(* Logix 5000 project; controller ACMI_PLC vendor 1 type 14 code 101 rev 19.11; software revision 19.01; part 3 of 18 *)

        [755].TIME.MICROSECOND := 993025, [755].EVENT := '2016/09/22   13:48:08   USER : PPS RESET FAULT BUTTON PRESSED', [756].TIME.YEAR := 2016, [756].TIME.MONTH := 9, [756].TIME.DAY := 22, [756].TIME.HOUR := 13, [756].TIME.MINUTE := 48, [756].TIME.SECOND := 37, [756].TIME.MICROSECOND := 592455, [756].EVENT := '2016/09/22   13:48:37   FAULT : QOW1 : Charge Outside Window Detected', [757].TIME.YEAR := 2016, [757].TIME.MONTH := 9, [757].TIME.DAY := 22, [757].TIME.HOUR := 13, [757].TIME.MINUTE := 58, [757].TIME.SECOND := 51, [757].TIME.MICROSECOND := 992497, [757].EVENT := '2016/09/22   13:58:51   USER : PPS RESET FAULT BUTTON PRESSED', [758].TIME.YEAR := 2016, [758].TIME.MONTH := 9, [758].TIME.DAY := 22, [758].TIME.HOUR := 13, [758].TIME.MINUTE := 59, [758].TIME.SECOND := 13, [758].TIME.MICROSECOND := 392501, [758].EVENT := '2016/09/22   13:59:13   USER : PPS RESET FAULT BUTTON PRESSED', [759].TIME.YEAR := 2016, [759].TIME.MONTH := 9, [759].TIME.DAY := 22, [759].TIME.HOUR := 14, [759].TIME.MINUTE := 6, [759].TIME.SECOND := 54, [759].TIME.MICROSECOND := 592461, [759].EVENT := '2016/09/22   14:06:54   FAULT : QOW1 : Charge Outside Window Detected', [760].TIME.YEAR := 2016, [760].TIME.MONTH := 9, [760].TIME.DAY := 22, [760].TIME.HOUR := 14, [760].TIME.MINUTE := 6, [760].TIME.SECOND := 54, [760].TIME.MICROSECOND := 692501, [760].EVENT := '2016/09/22   14:06:54   USER : PPS RESET FAULT BUTTON PRESSED', [761].TIME.YEAR := 2016, [761].TIME.MONTH := 9, [761].TIME.DAY := 22, [761].TIME.HOUR := 14, [761].TIME.MINUTE := 9, [761].TIME.SECOND := 18, [761].TIME.MICROSECOND := 892502, [761].EVENT := '2016/09/22   14:09:18   USER : PPS RESET FAULT BUTTON PRESSED', [762].TIME.YEAR := 2016, [762].TIME.MONTH := 9, [762].TIME.DAY := 22, [762].TIME.HOUR := 14, [762].TIME.MINUTE := 9, [762].TIME.SECOND := 19, [762].TIME.MICROSECOND := 92924, [762].EVENT := '2016/09/22   14:09:19   USER : PPS RESET FAULT BUTTON PRESSED', [763].TIME.YEAR := 2016, [763].TIME.MONTH := 9,
        [763].TIME.DAY := 22, [763].TIME.HOUR := 14, [763].TIME.MINUTE := 9, [763].TIME.SECOND := 19, [763].TIME.MICROSECOND := 292500, [763].EVENT := '2016/09/22   14:09:19   USER : PPS RESET FAULT BUTTON PRESSED', [764].TIME.YEAR := 2016, [764].TIME.MONTH := 9, [764].TIME.DAY := 22, [764].TIME.HOUR := 14, [764].TIME.MINUTE := 10, [764].TIME.SECOND := 9, [764].TIME.MICROSECOND := 92519, [764].EVENT := '2016/09/22   14:10:09   USER : PPS RESET FAULT BUTTON PRESSED', [765].TIME.YEAR := 2016, [765].TIME.MONTH := 9, [765].TIME.DAY := 22, [765].TIME.HOUR := 14, [765].TIME.MINUTE := 10, [765].TIME.SECOND := 22, [765].TIME.MICROSECOND := 892490, [765].EVENT := '2016/09/22   14:10:22   FAULT : QOW1 : Charge Outside Window Detected', [766].TIME.YEAR := 2016, [766].TIME.MONTH := 9, [766].TIME.DAY := 22, [766].TIME.HOUR := 14, [766].TIME.MINUTE := 14, [766].TIME.SECOND := 58, [766].TIME.MICROSECOND := 893026, [766].EVENT := '2016/09/22   14:14:58   USER : PPS RESET FAULT BUTTON PRESSED', [767].TIME.YEAR := 2016, [767].TIME.MONTH := 9, [767].TIME.DAY := 22, [767].TIME.HOUR := 14, [767].TIME.MINUTE := 17, [767].TIME.SECOND := 16, [767].TIME.MICROSECOND := 392944, [767].EVENT := '2016/09/22   14:17:16   USER : PPS RESET FAULT BUTTON PRESSED', [768].TIME.YEAR := 2016, [768].TIME.MONTH := 9, [768].TIME.DAY := 22, [768].TIME.HOUR := 14, [768].TIME.MINUTE := 24, [768].TIME.SECOND := 16, [768].TIME.MICROSECOND := 292454, [768].EVENT := '2016/09/22   14:24:16   FAULT : QOW1 : Charge Outside Window Detected', [769].TIME.YEAR := 2016, [769].TIME.MONTH := 9, [769].TIME.DAY := 22, [769].TIME.HOUR := 14, [769].TIME.MINUTE := 24, [769].TIME.SECOND := 16, [769].TIME.MICROSECOND := 492501, [769].EVENT := '2016/09/22   14:24:16   USER : PPS RESET FAULT BUTTON PRESSED', [770].TIME.YEAR := 2016, [770].TIME.MONTH := 9, [770].TIME.DAY := 22, [770].TIME.HOUR := 14, [770].TIME.MINUTE := 26, [770].TIME.SECOND := 11,
        [770].TIME.MICROSECOND := 293045, [770].EVENT := '2016/09/22   14:26:11   USER : PPS RESET FAULT BUTTON PRESSED', [771].TIME.YEAR := 2016, [771].TIME.MONTH := 9, [771].TIME.DAY := 22, [771].TIME.HOUR := 14, [771].TIME.MINUTE := 31, [771].TIME.SECOND := 56, [771].TIME.MICROSECOND := 692937, [771].EVENT := '2016/09/22   14:31:56   USER : PPS RESET FAULT BUTTON PRESSED', [772].TIME.YEAR := 2016, [772].TIME.MONTH := 9, [772].TIME.DAY := 22, [772].TIME.HOUR := 14, [772].TIME.MINUTE := 33, [772].TIME.SECOND := 35, [772].TIME.MICROSECOND := 92499, [772].EVENT := '2016/09/22   14:33:35   USER : PPS RESET FAULT BUTTON PRESSED', [773].TIME.YEAR := 2016, [773].TIME.MONTH := 9, [773].TIME.DAY := 22, [773].TIME.HOUR := 14, [773].TIME.MINUTE := 34, [773].TIME.SECOND := 33, [773].TIME.MICROSECOND := 892502, [773].EVENT := '2016/09/22   14:34:33   FAULT : QOW1 : Charge Outside Window Detected', [774].TIME.YEAR := 2016, [774].TIME.MONTH := 9, [774].TIME.DAY := 22, [774].TIME.HOUR := 14, [774].TIME.MINUTE := 44, [774].TIME.SECOND := 35, [774].TIME.MICROSECOND := 492454, [774].EVENT := '2016/09/22   14:44:35   FAULT : QOW1 : Charge Outside Window Detected', [775].TIME.YEAR := 2016, [775].TIME.MONTH := 9, [775].TIME.DAY := 22, [775].TIME.HOUR := 14, [775].TIME.MINUTE := 44, [775].TIME.SECOND := 35, [775].TIME.MICROSECOND := 793029, [775].EVENT := '2016/09/22   14:44:35   USER : PPS RESET FAULT BUTTON PRESSED', [776].TIME.YEAR := 2016, [776].TIME.MONTH := 9, [776].TIME.DAY := 22, [776].TIME.HOUR := 14, [776].TIME.MINUTE := 45, [776].TIME.SECOND := 20, [776].TIME.MICROSECOND := 292508, [776].EVENT := '2016/09/22   14:45:20   USER : PPS RESET FAULT BUTTON PRESSED', [777].TIME.YEAR := 2016, [777].TIME.MONTH := 9, [777].TIME.DAY := 22, [777].TIME.HOUR := 14, [777].TIME.MINUTE := 52, [777].TIME.SECOND := 30, [777].TIME.MICROSECOND := 192458, [777].EVENT := '2016/09/22   14:52:30   FAULT : QOW1 : Charge Outside Window Detected', [778].TIME.YEAR := 2016, [778].TIME.MONTH := 9,
        [778].TIME.DAY := 22, [778].TIME.HOUR := 14, [778].TIME.MINUTE := 52, [778].TIME.SECOND := 30, [778].TIME.MICROSECOND := 792503, [778].EVENT := '2016/09/22   14:52:30   USER : PPS RESET FAULT BUTTON PRESSED', [779].TIME.YEAR := 2016, [779].TIME.MONTH := 9, [779].TIME.DAY := 22, [779].TIME.HOUR := 14, [779].TIME.MINUTE := 54, [779].TIME.SECOND := 20, [779].TIME.MICROSECOND := 992503, [779].EVENT := '2016/09/22   14:54:20   USER : PPS RESET FAULT BUTTON PRESSED', [780].TIME.YEAR := 2016, [780].TIME.MONTH := 9, [780].TIME.DAY := 22, [780].TIME.HOUR := 14, [780].TIME.MINUTE := 54, [780].TIME.SECOND := 43, [780].TIME.MICROSECOND := 592930, [780].EVENT := '2016/09/22   14:54:43   USER : PPS RESET FAULT BUTTON PRESSED', [781].TIME.YEAR := 2016, [781].TIME.MONTH := 9, [781].TIME.DAY := 22, [781].TIME.HOUR := 14, [781].TIME.MINUTE := 59, [781].TIME.SECOND := 29, [781].TIME.MICROSECOND := 592463, [781].EVENT := '2016/09/22   14:59:29   FAULT : QOW1 : Charge Outside Window Detected', [782].TIME.YEAR := 2016, [782].TIME.MONTH := 9, [782].TIME.DAY := 22, [782].TIME.HOUR := 14, [782].TIME.MINUTE := 59, [782].TIME.SECOND := 29, [782].TIME.MICROSECOND := 893020, [782].EVENT := '2016/09/22   14:59:29   USER : PPS RESET FAULT BUTTON PRESSED', [783].TIME.YEAR := 2016, [783].TIME.MONTH := 9, [783].TIME.DAY := 22, [783].TIME.HOUR := 15, [783].TIME.MINUTE := 1, [783].TIME.SECOND := 30, [783].TIME.MICROSECOND := 992511, [783].EVENT := '2016/09/22   15:01:30   USER : PPS RESET FAULT BUTTON PRESSED', [784].TIME.YEAR := 2016, [784].TIME.MONTH := 9, [784].TIME.DAY := 22, [784].TIME.HOUR := 15, [784].TIME.MINUTE := 1, [784].TIME.SECOND := 35, [784].TIME.MICROSECOND := 392501, [784].EVENT := '2016/09/22   15:01:35   USER : PPS RESET FAULT BUTTON PRESSED', [785].TIME.YEAR := 2016, [785].TIME.MONTH := 9, [785].TIME.DAY := 22, [785].TIME.HOUR := 15, [785].TIME.MINUTE := 6, [785].TIME.SECOND := 4,
        [785].TIME.MICROSECOND := 392456, [785].EVENT := '2016/09/22   15:06:04   FAULT : QOW1 : Charge Outside Window Detected', [786].TIME.YEAR := 2016, [786].TIME.MONTH := 9, [786].TIME.DAY := 22, [786].TIME.HOUR := 15, [786].TIME.MINUTE := 6, [786].TIME.SECOND := 5, [786].TIME.MICROSECOND := 292497, [786].EVENT := '2016/09/22   15:06:05   USER : PPS RESET FAULT BUTTON PRESSED', [787].TIME.YEAR := 2016, [787].TIME.MONTH := 9, [787].TIME.DAY := 22, [787].TIME.HOUR := 15, [787].TIME.MINUTE := 8, [787].TIME.SECOND := 5, [787].TIME.MICROSECOND := 292503, [787].EVENT := '2016/09/22   15:08:05   USER : PPS RESET FAULT BUTTON PRESSED', [788].TIME.YEAR := 2016, [788].TIME.MONTH := 9, [788].TIME.DAY := 22, [788].TIME.HOUR := 15, [788].TIME.MINUTE := 8, [788].TIME.SECOND := 22, [788].TIME.MICROSECOND := 792884, [788].EVENT := '2016/09/22   15:08:22   FAULT : QOW1 : Charge Outside Window Detected', [789].TIME.YEAR := 2016, [789].TIME.MONTH := 9, [789].TIME.DAY := 22, [789].TIME.HOUR := 15, [789].TIME.MINUTE := 14, [789].TIME.SECOND := 51, [789].TIME.MICROSECOND := 392574, [789].EVENT := '2016/09/22   15:14:51   USER : PPS RESET FAULT BUTTON PRESSED', [790].TIME.YEAR := 2016, [790].TIME.MONTH := 9, [790].TIME.DAY := 22, [790].TIME.HOUR := 15, [790].TIME.MINUTE := 14, [790].TIME.SECOND := 53, [790].TIME.MICROSECOND := 892507, [790].EVENT := '2016/09/22   15:14:53   USER : PPS RESET FAULT BUTTON PRESSED', [791].TIME.YEAR := 2016, [791].TIME.MONTH := 9, [791].TIME.DAY := 22, [791].TIME.HOUR := 15, [791].TIME.MINUTE := 16, [791].TIME.SECOND := 15, [791].TIME.MICROSECOND := 692506, [791].EVENT := '2016/09/22   15:16:15   USER : PPS RESET FAULT BUTTON PRESSED', [792].TIME.YEAR := 2016, [792].TIME.MONTH := 9, [792].TIME.DAY := 22, [792].TIME.HOUR := 15, [792].TIME.MINUTE := 24, [792].TIME.SECOND := 17, [792].TIME.MICROSECOND := 92458, [792].EVENT := '2016/09/22   15:24:17   FAULT : QOW1 : Charge Outside Window Detected', [793].TIME.YEAR := 2016, [793].TIME.MONTH := 9,
        [793].TIME.DAY := 22, [793].TIME.HOUR := 15, [793].TIME.MINUTE := 24, [793].TIME.SECOND := 17, [793].TIME.MICROSECOND := 292502, [793].EVENT := '2016/09/22   15:24:17   USER : PPS RESET FAULT BUTTON PRESSED', [794].TIME.YEAR := 2016, [794].TIME.MONTH := 9, [794].TIME.DAY := 22, [794].TIME.HOUR := 15, [794].TIME.MINUTE := 25, [794].TIME.SECOND := 45, [794].TIME.MICROSECOND := 93021, [794].EVENT := '2016/09/22   15:25:45   USER : PPS RESET FAULT BUTTON PRESSED', [795].TIME.YEAR := 2016, [795].TIME.MONTH := 9, [795].TIME.DAY := 22, [795].TIME.HOUR := 15, [795].TIME.MINUTE := 27, [795].TIME.SECOND := 48, [795].TIME.MICROSECOND := 692501, [795].EVENT := '2016/09/22   15:27:48   USER : PPS RESET FAULT BUTTON PRESSED', [796].TIME.YEAR := 2016, [796].TIME.MONTH := 9, [796].TIME.DAY := 22, [796].TIME.HOUR := 15, [796].TIME.MINUTE := 27, [796].TIME.SECOND := 53, [796].TIME.MICROSECOND := 292498, [796].EVENT := '2016/09/22   15:27:53   USER : PPS RESET FAULT BUTTON PRESSED', [797].TIME.YEAR := 2016, [797].TIME.MONTH := 9, [797].TIME.DAY := 22, [797].TIME.HOUR := 15, [797].TIME.MINUTE := 28, [797].TIME.SECOND := 8, [797].TIME.MICROSECOND := 692887, [797].EVENT := '2016/09/22   15:28:08   FAULT : QOW1 : Charge Outside Window Detected', [798].TIME.YEAR := 2016, [798].TIME.MONTH := 9, [798].TIME.DAY := 22, [798].TIME.HOUR := 15, [798].TIME.MINUTE := 37, [798].TIME.SECOND := 46, [798].TIME.MICROSECOND := 92504, [798].EVENT := '2016/09/22   15:37:46   USER : PPS RESET FAULT BUTTON PRESSED', [799].TIME.YEAR := 2016, [799].TIME.MONTH := 9, [799].TIME.DAY := 22, [799].TIME.HOUR := 15, [799].TIME.MINUTE := 40, [799].TIME.SECOND := 5, [799].TIME.MICROSECOND := 692501, [799].EVENT := '2016/09/22   15:40:05   USER : PPS RESET FAULT BUTTON PRESSED', [800].TIME.YEAR := 2016, [800].TIME.MONTH := 9, [800].TIME.DAY := 22, [800].TIME.HOUR := 15, [800].TIME.MINUTE := 45, [800].TIME.MICROSECOND := 692496,
        [800].EVENT := '2016/09/22   15:45:00   USER : PPS RESET FAULT BUTTON PRESSED', [801].TIME.YEAR := 2016, [801].TIME.MONTH := 9, [801].TIME.DAY := 22, [801].TIME.HOUR := 15, [801].TIME.MINUTE := 48, [801].TIME.SECOND := 9, [801].TIME.MICROSECOND := 292507, [801].EVENT := '2016/09/22   15:48:09   USER : PPS RESET FAULT BUTTON PRESSED', [802].TIME.YEAR := 2016, [802].TIME.MONTH := 9, [802].TIME.DAY := 22, [802].TIME.HOUR := 15, [802].TIME.MINUTE := 48, [802].TIME.SECOND := 14, [802].TIME.MICROSECOND := 593026, [802].EVENT := '2016/09/22   15:48:14   USER : PPS RESET FAULT BUTTON PRESSED', [803].TIME.YEAR := 2016, [803].TIME.MONTH := 9, [803].TIME.DAY := 22, [803].TIME.HOUR := 15, [803].TIME.MINUTE := 53, [803].TIME.SECOND := 52, [803].TIME.MICROSECOND := 692453, [803].EVENT := '2016/09/22   15:53:52   FAULT : QOW1 : Charge Outside Window Detected', [804].TIME.YEAR := 2016, [804].TIME.MONTH := 9, [804].TIME.DAY := 22, [804].TIME.HOUR := 15, [804].TIME.MINUTE := 53, [804].TIME.SECOND := 52, [804].TIME.MICROSECOND := 992541, [804].EVENT := '2016/09/22   15:53:52   USER : PPS RESET FAULT BUTTON PRESSED', [805].TIME.YEAR := 2016, [805].TIME.MONTH := 9, [805].TIME.DAY := 22, [805].TIME.HOUR := 15, [805].TIME.MINUTE := 55, [805].TIME.SECOND := 30, [805].TIME.MICROSECOND := 292501, [805].EVENT := '2016/09/22   15:55:30   USER : PPS RESET FAULT BUTTON PRESSED', [806].TIME.YEAR := 2016, [806].TIME.MONTH := 9, [806].TIME.DAY := 22, [806].TIME.HOUR := 15, [806].TIME.MINUTE := 56, [806].TIME.SECOND := 39, [806].TIME.MICROSECOND := 92504, [806].EVENT := '2016/09/22   15:56:39   USER : PPS RESET FAULT BUTTON PRESSED', [807].TIME.YEAR := 2016, [807].TIME.MONTH := 9, [807].TIME.DAY := 22, [807].TIME.HOUR := 16, [807].TIME.SECOND := 24, [807].TIME.MICROSECOND := 592887, [807].EVENT := '2016/09/22   16:00:24   FAULT : QOW1 : Charge Outside Window Detected', [808].TIME.YEAR := 2016, [808].TIME.MONTH := 9, [808].TIME.DAY := 22, [808].TIME.HOUR := 16,
        [808].TIME.SECOND := 25, [808].TIME.MICROSECOND := 92935, [808].EVENT := '2016/09/22   16:00:25   USER : PPS RESET FAULT BUTTON PRESSED', [809].TIME.YEAR := 2016, [809].TIME.MONTH := 9, [809].TIME.DAY := 22, [809].TIME.HOUR := 16, [809].TIME.MINUTE := 2, [809].TIME.SECOND := 43, [809].TIME.MICROSECOND := 692936, [809].EVENT := '2016/09/22   16:02:43   USER : PPS RESET FAULT BUTTON PRESSED', [810].TIME.YEAR := 2016, [810].TIME.MONTH := 9, [810].TIME.DAY := 22, [810].TIME.HOUR := 16, [810].TIME.MINUTE := 4, [810].TIME.SECOND := 4, [810].TIME.MICROSECOND := 792503, [810].EVENT := '2016/09/22   16:04:04   USER : PPS RESET FAULT BUTTON PRESSED', [811].TIME.YEAR := 2016, [811].TIME.MONTH := 9, [811].TIME.DAY := 22, [811].TIME.HOUR := 16, [811].TIME.MINUTE := 4, [811].TIME.SECOND := 14, [811].TIME.MICROSECOND := 192460, [811].EVENT := '2016/09/22   16:04:14   FAULT : QOW1 : Charge Outside Window Detected', [812].TIME.YEAR := 2016, [812].TIME.MONTH := 9, [812].TIME.DAY := 22, [812].TIME.HOUR := 16, [812].TIME.MINUTE := 13, [812].TIME.SECOND := 37, [812].TIME.MICROSECOND := 992500, [812].EVENT := '2016/09/22   16:13:37   USER : PPS RESET FAULT BUTTON PRESSED', [813].TIME.YEAR := 2016, [813].TIME.MONTH := 9, [813].TIME.DAY := 22, [813].TIME.HOUR := 16, [813].TIME.MINUTE := 15, [813].TIME.SECOND := 18, [813].TIME.MICROSECOND := 492646, [813].EVENT := '2016/09/22   16:15:18   USER : PPS RESET FAULT BUTTON PRESSED', [814].TIME.YEAR := 2016, [814].TIME.MONTH := 9, [814].TIME.DAY := 22, [814].TIME.HOUR := 16, [814].TIME.MINUTE := 19, [814].TIME.SECOND := 56, [814].TIME.MICROSECOND := 592459, [814].EVENT := '2016/09/22   16:19:56   FAULT : QOW1 : Charge Outside Window Detected', [815].TIME.YEAR := 2016, [815].TIME.MONTH := 9, [815].TIME.DAY := 22, [815].TIME.HOUR := 16, [815].TIME.MINUTE := 19, [815].TIME.SECOND := 56, [815].TIME.MICROSECOND := 792506, [815].EVENT := '2016/09/22   16:19:56   USER : PPS RESET FAULT BUTTON PRESSED', [816].TIME.YEAR := 2016,
        [816].TIME.MONTH := 9, [816].TIME.DAY := 22, [816].TIME.HOUR := 16, [816].TIME.MINUTE := 21, [816].TIME.SECOND := 32, [816].TIME.MICROSECOND := 892505, [816].EVENT := '2016/09/22   16:21:32   USER : PPS RESET FAULT BUTTON PRESSED', [817].TIME.YEAR := 2016, [817].TIME.MONTH := 9, [817].TIME.DAY := 22, [817].TIME.HOUR := 16, [817].TIME.MINUTE := 25, [817].TIME.SECOND := 22, [817].TIME.MICROSECOND := 992455, [817].EVENT := '2016/09/22   16:25:22   FAULT : QOW1 : Charge Outside Window Detected', [818].TIME.YEAR := 2016, [818].TIME.MONTH := 9, [818].TIME.DAY := 22, [818].TIME.HOUR := 16, [818].TIME.MINUTE := 25, [818].TIME.SECOND := 23, [818].TIME.MICROSECOND := 92503, [818].EVENT := '2016/09/22   16:25:23   USER : PPS RESET FAULT BUTTON PRESSED', [819].TIME.YEAR := 2016, [819].TIME.MONTH := 9, [819].TIME.DAY := 22, [819].TIME.HOUR := 16, [819].TIME.MINUTE := 26, [819].TIME.SECOND := 55, [819].TIME.MICROSECOND := 492497, [819].EVENT := '2016/09/22   16:26:55   USER : PPS RESET FAULT BUTTON PRESSED', [820].TIME.YEAR := 2016, [820].TIME.MONTH := 9, [820].TIME.DAY := 22, [820].TIME.HOUR := 16, [820].TIME.MINUTE := 27, [820].TIME.SECOND := 39, [820].TIME.MICROSECOND := 992977, [820].EVENT := '2016/09/22   16:27:39   FAULT : QOW1 : Charge Outside Window Detected', [821].TIME.YEAR := 2016, [821].TIME.MONTH := 9, [821].TIME.DAY := 22, [821].TIME.HOUR := 16, [821].TIME.MINUTE := 31, [821].TIME.SECOND := 17, [821].TIME.MICROSECOND := 993097, [821].EVENT := '2016/09/22   16:31:17   USER : PPS RESET FAULT BUTTON PRESSED', [822].TIME.YEAR := 2016, [822].TIME.MONTH := 9, [822].TIME.DAY := 22, [822].TIME.HOUR := 16, [822].TIME.MINUTE := 32, [822].TIME.SECOND := 41, [822].TIME.MICROSECOND := 92499, [822].EVENT := '2016/09/22   16:32:41   USER : PPS RESET FAULT BUTTON PRESSED', [823].TIME.YEAR := 2016, [823].TIME.MONTH := 9, [823].TIME.DAY := 22, [823].TIME.HOUR := 16, [823].TIME.MINUTE := 33,
        [823].TIME.SECOND := 17, [823].TIME.MICROSECOND := 192884, [823].EVENT := '2016/09/22   16:33:17   FAULT : QOW1 : Charge Outside Window Detected', [824].TIME.YEAR := 2016, [824].TIME.MONTH := 9, [824].TIME.DAY := 22, [824].TIME.HOUR := 16, [824].TIME.MINUTE := 36, [824].TIME.SECOND := 37, [824].TIME.MICROSECOND := 292508, [824].EVENT := '2016/09/22   16:36:37   USER : PPS RESET FAULT BUTTON PRESSED', [825].TIME.YEAR := 2016, [825].TIME.MONTH := 9, [825].TIME.DAY := 22, [825].TIME.HOUR := 16, [825].TIME.MINUTE := 38, [825].TIME.SECOND := 11, [825].TIME.MICROSECOND := 292506, [825].EVENT := '2016/09/22   16:38:11   USER : PPS RESET FAULT BUTTON PRESSED', [826].TIME.YEAR := 2016, [826].TIME.MONTH := 9, [826].TIME.DAY := 22, [826].TIME.HOUR := 16, [826].TIME.MINUTE := 39, [826].TIME.SECOND := 9, [826].TIME.MICROSECOND := 193027, [826].EVENT := '2016/09/22   16:39:09   USER : PPS RESET FAULT BUTTON PRESSED', [827].TIME.YEAR := 2016, [827].TIME.MONTH := 9, [827].TIME.DAY := 22, [827].TIME.HOUR := 16, [827].TIME.MINUTE := 39, [827].TIME.SECOND := 17, [827].TIME.MICROSECOND := 892887, [827].EVENT := '2016/09/22   16:39:17   FAULT : QOW1 : Charge Outside Window Detected', [828].TIME.YEAR := 2016, [828].TIME.MONTH := 9, [828].TIME.DAY := 22, [828].TIME.HOUR := 16, [828].TIME.MINUTE := 46, [828].TIME.SECOND := 29, [828].TIME.MICROSECOND := 192503, [828].EVENT := '2016/09/22   16:46:29   USER : PPS RESET FAULT BUTTON PRESSED', [829].TIME.YEAR := 2016, [829].TIME.MONTH := 9, [829].TIME.DAY := 22, [829].TIME.HOUR := 16, [829].TIME.MINUTE := 46, [829].TIME.SECOND := 44, [829].TIME.MICROSECOND := 292544, [829].EVENT := '2016/09/22   16:46:44   USER : PPS RESET FAULT BUTTON PRESSED', [830].TIME.YEAR := 2016, [830].TIME.MONTH := 9, [830].TIME.DAY := 22, [830].TIME.HOUR := 16, [830].TIME.MINUTE := 48, [830].TIME.SECOND := 42, [830].TIME.MICROSECOND := 992499, [830].EVENT := '2016/09/22   16:48:42   USER : PPS RESET FAULT BUTTON PRESSED', [831].TIME.YEAR := 2016,
        [831].TIME.MONTH := 9, [831].TIME.DAY := 22, [831].TIME.HOUR := 16, [831].TIME.MINUTE := 57, [831].TIME.SECOND := 35, [831].TIME.MICROSECOND := 992503, [831].EVENT := '2016/09/22   16:57:35   USER : PPS RESET FAULT BUTTON PRESSED', [832].TIME.YEAR := 2016, [832].TIME.MONTH := 9, [832].TIME.DAY := 22, [832].TIME.HOUR := 17, [832].TIME.MINUTE := 6, [832].TIME.MICROSECOND := 992512, [832].EVENT := '2016/09/22   17:06:00   USER : PPS RESET FAULT BUTTON PRESSED', [833].TIME.YEAR := 2016, [833].TIME.MONTH := 9, [833].TIME.DAY := 22, [833].TIME.HOUR := 17, [833].TIME.MINUTE := 12, [833].TIME.SECOND := 42, [833].TIME.MICROSECOND := 192573, [833].EVENT := '2016/09/22   17:12:42   FAULT : QOW1 : Charge Outside Window Detected', [834].TIME.YEAR := 2016, [834].TIME.MONTH := 9, [834].TIME.DAY := 22, [834].TIME.HOUR := 17, [834].TIME.MINUTE := 13, [834].TIME.SECOND := 36, [834].TIME.MICROSECOND := 992648, [834].EVENT := '2016/09/22   17:13:36   USER : PPS RESET FAULT BUTTON PRESSED', [835].TIME.YEAR := 2016, [835].TIME.MONTH := 9, [835].TIME.DAY := 22, [835].TIME.HOUR := 17, [835].TIME.MINUTE := 14, [835].TIME.SECOND := 24, [835].TIME.MICROSECOND := 792499, [835].EVENT := '2016/09/22   17:14:24   USER : PPS RESET FAULT BUTTON PRESSED', [836].TIME.YEAR := 2016, [836].TIME.MONTH := 9, [836].TIME.DAY := 22, [836].TIME.HOUR := 17, [836].TIME.MINUTE := 14, [836].TIME.SECOND := 44, [836].TIME.MICROSECOND := 992504, [836].EVENT := '2016/09/22   17:14:44   USER : PPS RESET FAULT BUTTON PRESSED', [837].TIME.YEAR := 2016, [837].TIME.MONTH := 9, [837].TIME.DAY := 22, [837].TIME.HOUR := 17, [837].TIME.MINUTE := 14, [837].TIME.SECOND := 54, [837].TIME.MICROSECOND := 592504, [837].EVENT := '2016/09/22   17:14:54   USER : PPS RESET FAULT BUTTON PRESSED', [838].TIME.YEAR := 2016, [838].TIME.MONTH := 9, [838].TIME.DAY := 22, [838].TIME.HOUR := 17, [838].TIME.MINUTE := 15, [838].TIME.SECOND := 24,
        [838].TIME.MICROSECOND := 192641, [838].EVENT := '2016/09/22   17:15:24   USER : PPS RESET FAULT BUTTON PRESSED', [839].TIME.YEAR := 2016, [839].TIME.MONTH := 9, [839].TIME.DAY := 22, [839].TIME.HOUR := 17, [839].TIME.MINUTE := 15, [839].TIME.SECOND := 48, [839].TIME.MICROSECOND := 192539, [839].EVENT := '2016/09/22   17:15:48   USER : PPS RESET FAULT BUTTON PRESSED', [840].TIME.YEAR := 2016, [840].TIME.MONTH := 9, [840].TIME.DAY := 22, [840].TIME.HOUR := 17, [840].TIME.MINUTE := 16, [840].TIME.SECOND := 12, [840].TIME.MICROSECOND := 992935, [840].EVENT := '2016/09/22   17:16:12   USER : PPS RESET FAULT BUTTON PRESSED', [841].TIME.YEAR := 2016, [841].TIME.MONTH := 9, [841].TIME.DAY := 22, [841].TIME.HOUR := 17, [841].TIME.MINUTE := 16, [841].TIME.SECOND := 14, [841].TIME.MICROSECOND := 692499, [841].EVENT := '2016/09/22   17:16:14   USER : PPS RESET FAULT BUTTON PRESSED', [842].TIME.YEAR := 2016, [842].TIME.MONTH := 9, [842].TIME.DAY := 22, [842].TIME.HOUR := 17, [842].TIME.MINUTE := 16, [842].TIME.SECOND := 40, [842].TIME.MICROSECOND := 192503, [842].EVENT := '2016/09/22   17:16:40   USER : PPS RESET FAULT BUTTON PRESSED', [843].TIME.YEAR := 2016, [843].TIME.MONTH := 9, [843].TIME.DAY := 22, [843].TIME.HOUR := 17, [843].TIME.MINUTE := 17, [843].TIME.SECOND := 4, [843].TIME.MICROSECOND := 92498, [843].EVENT := '2016/09/22   17:17:04   USER : PPS RESET FAULT BUTTON PRESSED', [844].TIME.YEAR := 2016, [844].TIME.MONTH := 9, [844].TIME.DAY := 22, [844].TIME.HOUR := 17, [844].TIME.MINUTE := 17, [844].TIME.SECOND := 22, [844].TIME.MICROSECOND := 692713, [844].EVENT := '2016/09/22   17:17:22   USER : PPS RESET FAULT BUTTON PRESSED', [845].TIME.YEAR := 2016, [845].TIME.MONTH := 9, [845].TIME.DAY := 22, [845].TIME.HOUR := 17, [845].TIME.MINUTE := 17, [845].TIME.SECOND := 23, [845].TIME.MICROSECOND := 392513, [845].EVENT := '2016/09/22   17:17:23   USER : PPS RESET FAULT BUTTON PRESSED', [846].TIME.YEAR := 2016, [846].TIME.MONTH := 9,
        [846].TIME.DAY := 22, [846].TIME.HOUR := 17, [846].TIME.MINUTE := 17, [846].TIME.SECOND := 27, [846].TIME.MICROSECOND := 893029, [846].EVENT := '2016/09/22   17:17:27   USER : PPS RESET FAULT BUTTON PRESSED', [847].TIME.YEAR := 2016, [847].TIME.MONTH := 9, [847].TIME.DAY := 22, [847].TIME.HOUR := 17, [847].TIME.MINUTE := 18, [847].TIME.SECOND := 1, [847].TIME.MICROSECOND := 92520, [847].EVENT := '2016/09/22   17:18:01   USER : PPS RESET FAULT BUTTON PRESSED', [848].TIME.YEAR := 2016, [848].TIME.MONTH := 9, [848].TIME.DAY := 22, [848].TIME.HOUR := 17, [848].TIME.MINUTE := 18, [848].TIME.SECOND := 18, [848].TIME.MICROSECOND := 793030, [848].EVENT := '2016/09/22   17:18:18   USER : PPS RESET FAULT BUTTON PRESSED', [849].TIME.YEAR := 2016, [849].TIME.MONTH := 9, [849].TIME.DAY := 22, [849].TIME.HOUR := 17, [849].TIME.MINUTE := 18, [849].TIME.SECOND := 36, [849].TIME.MICROSECOND := 792498, [849].EVENT := '2016/09/22   17:18:36   USER : PPS RESET FAULT BUTTON PRESSED', [850].TIME.YEAR := 2016, [850].TIME.MONTH := 9, [850].TIME.DAY := 22, [850].TIME.HOUR := 17, [850].TIME.MINUTE := 19, [850].TIME.SECOND := 19, [850].TIME.MICROSECOND := 492502, [850].EVENT := '2016/09/22   17:19:19   USER : PPS RESET FAULT BUTTON PRESSED', [851].TIME.YEAR := 2016, [851].TIME.MONTH := 9, [851].TIME.DAY := 23, [851].TIME.HOUR := 9, [851].TIME.MINUTE := 49, [851].TIME.SECOND := 56, [851].TIME.MICROSECOND := 692502, [851].EVENT := '2016/09/23   09:49:56   USER : PPS RESET FAULT BUTTON PRESSED', [852].TIME.YEAR := 2016, [852].TIME.MONTH := 9, [852].TIME.DAY := 23, [852].TIME.HOUR := 9, [852].TIME.MINUTE := 51, [852].TIME.SECOND := 27, [852].TIME.MICROSECOND := 93021, [852].EVENT := '2016/09/23   09:51:27   USER : PPS RESET FAULT BUTTON PRESSED', [853].TIME.YEAR := 2016, [853].TIME.MONTH := 9, [853].TIME.DAY := 23, [853].TIME.HOUR := 9, [853].TIME.MINUTE := 55, [853].TIME.SECOND := 7,
        [853].TIME.MICROSECOND := 992505, [853].EVENT := '2016/09/23   09:55:07   USER : PPS RESET FAULT BUTTON PRESSED', [854].TIME.YEAR := 2016, [854].TIME.MONTH := 9, [854].TIME.DAY := 23, [854].TIME.HOUR := 14, [854].TIME.MINUTE := 51, [854].TIME.SECOND := 16, [854].TIME.MICROSECOND := 892451, [854].EVENT := '2016/09/23   14:51:16   FAULT : QOW1 : Charge Outside Window Detected', [855].TIME.YEAR := 2016, [855].TIME.MONTH := 9, [855].TIME.DAY := 23, [855].TIME.HOUR := 14, [855].TIME.MINUTE := 51, [855].TIME.SECOND := 17, [855].TIME.MICROSECOND := 92498, [855].EVENT := '2016/09/23   14:51:17   USER : PPS RESET FAULT BUTTON PRESSED', [856].TIME.YEAR := 2016, [856].TIME.MONTH := 9, [856].TIME.DAY := 23, [856].TIME.HOUR := 14, [856].TIME.MINUTE := 55, [856].TIME.SECOND := 53, [856].TIME.MICROSECOND := 293149, [856].EVENT := '2016/09/23   14:55:53   USER : PPS RESET FAULT BUTTON PRESSED', [857].TIME.YEAR := 2016, [857].TIME.MONTH := 9, [857].TIME.DAY := 23, [857].TIME.HOUR := 15, [857].TIME.MINUTE := 9, [857].TIME.SECOND := 48, [857].TIME.MICROSECOND := 392456, [857].EVENT := '2016/09/23   15:09:48   FAULT : QOW1 : Charge Outside Window Detected', [858].TIME.YEAR := 2016, [858].TIME.MONTH := 9, [858].TIME.DAY := 23, [858].TIME.HOUR := 15, [858].TIME.MINUTE := 9, [858].TIME.SECOND := 48, [858].TIME.MICROSECOND := 592506, [858].EVENT := '2016/09/23   15:09:48   USER : PPS RESET FAULT BUTTON PRESSED', [859].TIME.YEAR := 2016, [859].TIME.MONTH := 9, [859].TIME.DAY := 23, [859].TIME.HOUR := 15, [859].TIME.MINUTE := 11, [859].TIME.SECOND := 50, [859].TIME.MICROSECOND := 592928, [859].EVENT := '2016/09/23   15:11:50   USER : PPS RESET FAULT BUTTON PRESSED', [860].TIME.YEAR := 2016, [860].TIME.MONTH := 9, [860].TIME.DAY := 23, [860].TIME.HOUR := 15, [860].TIME.MINUTE := 12, [860].TIME.SECOND := 20, [860].TIME.MICROSECOND := 692500, [860].EVENT := '2016/09/23   15:12:20   USER : PPS RESET FAULT BUTTON PRESSED', [861].TIME.YEAR := 2016, [861].TIME.MONTH := 9,
        [861].TIME.DAY := 23, [861].TIME.HOUR := 15, [861].TIME.MINUTE := 12, [861].TIME.SECOND := 23, [861].TIME.MICROSECOND := 892504, [861].EVENT := '2016/09/23   15:12:23   USER : PPS RESET FAULT BUTTON PRESSED', [862].TIME.YEAR := 2016, [862].TIME.MONTH := 9, [862].TIME.DAY := 23, [862].TIME.HOUR := 15, [862].TIME.MINUTE := 12, [862].TIME.SECOND := 24, [862].TIME.MICROSECOND := 193017, [862].EVENT := '2016/09/23   15:12:24   USER : PPS RESET FAULT BUTTON PRESSED', [863].TIME.YEAR := 2016, [863].TIME.MONTH := 9, [863].TIME.DAY := 23, [863].TIME.HOUR := 15, [863].TIME.MINUTE := 13, [863].TIME.SECOND := 20, [863].TIME.MICROSECOND := 792504, [863].EVENT := '2016/09/23   15:13:20   USER : PPS RESET FAULT BUTTON PRESSED', [864].TIME.YEAR := 2016, [864].TIME.MONTH := 9, [864].TIME.DAY := 23, [864].TIME.HOUR := 15, [864].TIME.MINUTE := 13, [864].TIME.SECOND := 36, [864].TIME.MICROSECOND := 392510, [864].EVENT := '2016/09/23   15:13:36   USER : PPS RESET FAULT BUTTON PRESSED', [865].TIME.YEAR := 2016, [865].TIME.MONTH := 9, [865].TIME.DAY := 23, [865].TIME.HOUR := 15, [865].TIME.MINUTE := 14, [865].TIME.SECOND := 4, [865].TIME.MICROSECOND := 493024, [865].EVENT := '2016/09/23   15:14:04   USER : PPS RESET FAULT BUTTON PRESSED', [866].TIME.YEAR := 2016, [866].TIME.MONTH := 9, [866].TIME.DAY := 23, [866].TIME.HOUR := 15, [866].TIME.MINUTE := 14, [866].TIME.SECOND := 20, [866].TIME.MICROSECOND := 492520, [866].EVENT := '2016/09/23   15:14:20   USER : PPS RESET FAULT BUTTON PRESSED', [867].TIME.YEAR := 2016, [867].TIME.MONTH := 9, [867].TIME.DAY := 23, [867].TIME.HOUR := 15, [867].TIME.MINUTE := 14, [867].TIME.SECOND := 38, [867].TIME.MICROSECOND := 692971, [867].EVENT := '2016/09/23   15:14:38   FAULT : QOW1 : Charge Outside Window Detected', [868].TIME.YEAR := 2016, [868].TIME.MONTH := 9, [868].TIME.DAY := 23, [868].TIME.HOUR := 15, [868].TIME.MINUTE := 16, [868].TIME.SECOND := 27,
        [868].TIME.MICROSECOND := 892500, [868].EVENT := '2016/09/23   15:16:27   USER : PPS RESET FAULT BUTTON PRESSED', [869].TIME.YEAR := 2016, [869].TIME.MONTH := 9, [869].TIME.DAY := 23, [869].TIME.HOUR := 15, [869].TIME.MINUTE := 44, [869].TIME.SECOND := 56, [869].TIME.MICROSECOND := 692501, [869].EVENT := '2016/09/23   15:44:56   USER : PPS RESET FAULT BUTTON PRESSED', [870].TIME.YEAR := 2016, [870].TIME.MONTH := 9, [870].TIME.DAY := 23, [870].TIME.HOUR := 15, [870].TIME.MINUTE := 46, [870].TIME.MICROSECOND := 692500, [870].EVENT := '2016/09/23   15:46:00   USER : PPS RESET FAULT BUTTON PRESSED', [871].TIME.YEAR := 2016, [871].TIME.MONTH := 9, [871].TIME.DAY := 23, [871].TIME.HOUR := 15, [871].TIME.MINUTE := 48, [871].TIME.SECOND := 24, [871].TIME.MICROSECOND := 592453, [871].EVENT := '2016/09/23   15:48:24   FAULT : QOW1 : Charge Outside Window Detected', [872].TIME.YEAR := 2016, [872].TIME.MONTH := 9, [872].TIME.DAY := 23, [872].TIME.HOUR := 15, [872].TIME.MINUTE := 48, [872].TIME.SECOND := 25, [872].TIME.MICROSECOND := 92500, [872].EVENT := '2016/09/23   15:48:25   USER : PPS RESET FAULT BUTTON PRESSED', [873].TIME.YEAR := 2016, [873].TIME.MONTH := 9, [873].TIME.DAY := 23, [873].TIME.HOUR := 15, [873].TIME.MINUTE := 48, [873].TIME.SECOND := 30, [873].TIME.MICROSECOND := 492554, [873].EVENT := '2016/09/23   15:48:30   USER : PPS RESET FAULT BUTTON PRESSED', [874].TIME.YEAR := 2016, [874].TIME.MONTH := 9, [874].TIME.DAY := 23, [874].TIME.HOUR := 15, [874].TIME.MINUTE := 50, [874].TIME.SECOND := 44, [874].TIME.MICROSECOND := 492501, [874].EVENT := '2016/09/23   15:50:44   USER : PPS RESET FAULT BUTTON PRESSED', [875].TIME.YEAR := 2016, [875].TIME.MONTH := 9, [875].TIME.DAY := 23, [875].TIME.HOUR := 15, [875].TIME.MINUTE := 51, [875].TIME.SECOND := 36, [875].TIME.MICROSECOND := 992498, [875].EVENT := '2016/09/23   15:51:36   USER : PPS RESET FAULT BUTTON PRESSED', [876].TIME.YEAR := 2016, [876].TIME.MONTH := 9, [876].TIME.DAY := 23,
        [876].TIME.HOUR := 15, [876].TIME.MINUTE := 51, [876].TIME.SECOND := 39, [876].TIME.MICROSECOND := 692501, [876].EVENT := '2016/09/23   15:51:39   USER : PPS RESET FAULT BUTTON PRESSED', [877].TIME.YEAR := 2016, [877].TIME.MONTH := 9, [877].TIME.DAY := 23, [877].TIME.HOUR := 15, [877].TIME.MINUTE := 51, [877].TIME.SECOND := 41, [877].TIME.MICROSECOND := 692505, [877].EVENT := '2016/09/23   15:51:41   USER : PPS RESET FAULT BUTTON PRESSED', [878].TIME.YEAR := 2016, [878].TIME.MONTH := 9, [878].TIME.DAY := 23, [878].TIME.HOUR := 15, [878].TIME.MINUTE := 52, [878].TIME.SECOND := 48, [878].TIME.MICROSECOND := 192459, [878].EVENT := '2016/09/23   15:52:48   FAULT : QOW1 : Charge Outside Window Detected', [879].TIME.YEAR := 2016, [879].TIME.MONTH := 9, [879].TIME.DAY := 23, [879].TIME.HOUR := 16, [879].TIME.MINUTE := 2, [879].TIME.SECOND := 55, [879].TIME.MICROSECOND := 92502, [879].EVENT := '2016/09/23   16:02:55   USER : PPS RESET FAULT BUTTON PRESSED', [880].TIME.YEAR := 2016, [880].TIME.MONTH := 9, [880].TIME.DAY := 23, [880].TIME.HOUR := 16, [880].TIME.MINUTE := 3, [880].TIME.SECOND := 3, [880].TIME.MICROSECOND := 992940, [880].EVENT := '2016/09/23   16:03:03   USER : PPS RESET FAULT BUTTON PRESSED', [881].TIME.YEAR := 2016, [881].TIME.MONTH := 9, [881].TIME.DAY := 23, [881].TIME.HOUR := 16, [881].TIME.MINUTE := 4, [881].TIME.SECOND := 44, [881].TIME.MICROSECOND := 592516, [881].EVENT := '2016/09/23   16:04:44   USER : PPS RESET FAULT BUTTON PRESSED', [882].TIME.YEAR := 2016, [882].TIME.MONTH := 9, [882].TIME.DAY := 23, [882].TIME.HOUR := 16, [882].TIME.MINUTE := 11, [882].TIME.SECOND := 4, [882].TIME.MICROSECOND := 192503, [882].EVENT := '2016/09/23   16:11:04   USER : PPS RESET FAULT BUTTON PRESSED', [883].TIME.YEAR := 2016, [883].TIME.MONTH := 9, [883].TIME.DAY := 23, [883].TIME.HOUR := 17, [883].TIME.MINUTE := 4, [883].TIME.SECOND := 39, [883].TIME.MICROSECOND := 492454,
        [883].EVENT := '2016/09/23   17:04:39   FAULT : QOW1 : Charge Outside Window Detected', [884].TIME.YEAR := 2016, [884].TIME.MONTH := 9, [884].TIME.DAY := 23, [884].TIME.HOUR := 17, [884].TIME.MINUTE := 4, [884].TIME.SECOND := 39, [884].TIME.MICROSECOND := 692516, [884].EVENT := '2016/09/23   17:04:39   USER : PPS RESET FAULT BUTTON PRESSED', [885].TIME.YEAR := 2016, [885].TIME.MONTH := 9, [885].TIME.DAY := 23, [885].TIME.HOUR := 17, [885].TIME.MINUTE := 18, [885].TIME.SECOND := 59, [885].TIME.MICROSECOND := 392456, [885].EVENT := '2016/09/23   17:18:59   FAULT : QOW1 : Charge Outside Window Detected', [886].TIME.YEAR := 2016, [886].TIME.MONTH := 9, [886].TIME.DAY := 23, [886].TIME.HOUR := 17, [886].TIME.MINUTE := 18, [886].TIME.SECOND := 59, [886].TIME.MICROSECOND := 592501, [886].EVENT := '2016/09/23   17:18:59   USER : PPS RESET FAULT BUTTON PRESSED', [887].TIME.YEAR := 2016, [887].TIME.MONTH := 9, [887].TIME.DAY := 23, [887].TIME.HOUR := 17, [887].TIME.MINUTE := 20, [887].TIME.SECOND := 2, [887].TIME.MICROSECOND := 992501, [887].EVENT := '2016/09/23   17:20:02   USER : PPS RESET FAULT BUTTON PRESSED', [888].TIME.YEAR := 2016, [888].TIME.MONTH := 9, [888].TIME.DAY := 24, [888].TIME.HOUR := 8, [888].TIME.MINUTE := 3, [888].TIME.SECOND := 22, [888].TIME.MICROSECOND := 492496, [888].EVENT := '2016/09/24   08:03:22   USER : PPS RESET FAULT BUTTON PRESSED', [889].TIME.YEAR := 2016, [889].TIME.MONTH := 9, [889].TIME.DAY := 24, [889].TIME.HOUR := 9, [889].TIME.MINUTE := 1, [889].TIME.SECOND := 56, [889].TIME.MICROSECOND := 592501, [889].EVENT := '2016/09/24   09:01:56   USER : PPS RESET FAULT BUTTON PRESSED', [890].TIME.YEAR := 2016, [890].TIME.MONTH := 9, [890].TIME.DAY := 24, [890].TIME.HOUR := 18, [890].TIME.MINUTE := 41, [890].TIME.MICROSECOND := 992499, [890].EVENT := '2016/09/24   18:41:00   USER : PPS RESET FAULT BUTTON PRESSED', [891].TIME.YEAR := 2016, [891].TIME.MONTH := 9, [891].TIME.DAY := 24, [891].TIME.HOUR := 18,
        [891].TIME.MINUTE := 44, [891].TIME.SECOND := 12, [891].TIME.MICROSECOND := 892502, [891].EVENT := '2016/09/24   18:44:12   USER : PPS RESET FAULT BUTTON PRESSED', [892].TIME.YEAR := 2016, [892].TIME.MONTH := 9, [892].TIME.DAY := 26, [892].TIME.HOUR := 1, [892].TIME.MINUTE := 53, [892].TIME.SECOND := 36, [892].TIME.MICROSECOND := 292450, [892].EVENT := '2016/09/26   01:53:36   FAULT : QOW1 : Charge Outside Window Detected', [893].TIME.YEAR := 2016, [893].TIME.MONTH := 9, [893].TIME.DAY := 26, [893].TIME.HOUR := 1, [893].TIME.MINUTE := 54, [893].TIME.SECOND := 55, [893].TIME.MICROSECOND := 592504, [893].EVENT := '2016/09/26   01:54:55   USER : PPS RESET FAULT BUTTON PRESSED', [894].TIME.YEAR := 2016, [894].TIME.MONTH := 9, [894].TIME.DAY := 26, [894].TIME.HOUR := 13, [894].TIME.MINUTE := 40, [894].TIME.SECOND := 20, [894].TIME.MICROSECOND := 93019, [894].EVENT := '2016/09/26   13:40:20   USER : PPS RESET FAULT BUTTON PRESSED', [895].TIME.YEAR := 2016, [895].TIME.MONTH := 9, [895].TIME.DAY := 26, [895].TIME.HOUR := 13, [895].TIME.MINUTE := 40, [895].TIME.SECOND := 23, [895].TIME.MICROSECOND := 192946, [895].EVENT := '2016/09/26   13:40:23   USER : PPS RESET FAULT BUTTON PRESSED', [896].TIME.YEAR := 2016, [896].TIME.MONTH := 9, [896].TIME.DAY := 26, [896].TIME.HOUR := 14, [896].TIME.MINUTE := 4, [896].TIME.SECOND := 11, [896].TIME.MICROSECOND := 692459, [896].EVENT := '2016/09/26   14:04:11   FAULT : QOW1 : Charge Outside Window Detected', [897].TIME.YEAR := 2016, [897].TIME.MONTH := 9, [897].TIME.DAY := 26, [897].TIME.HOUR := 14, [897].TIME.MINUTE := 16, [897].TIME.SECOND := 43, [897].TIME.MICROSECOND := 592502, [897].EVENT := '2016/09/26   14:16:43   USER : PPS RESET FAULT BUTTON PRESSED', [898].TIME.YEAR := 2016, [898].TIME.MONTH := 9, [898].TIME.DAY := 26, [898].TIME.HOUR := 14, [898].TIME.MINUTE := 16, [898].TIME.SECOND := 46, [898].TIME.MICROSECOND := 592495, [898].EVENT := '2016/09/26   14:16:46   USER : PPS RESET FAULT BUTTON PRESSED',
        [899].TIME.YEAR := 2016, [899].TIME.MONTH := 9, [899].TIME.DAY := 26, [899].TIME.HOUR := 14, [899].TIME.MINUTE := 23, [899].TIME.SECOND := 5, [899].TIME.MICROSECOND := 392452, [899].EVENT := '2016/09/26   14:23:05   FAULT : WDT : Trigger Rate LOW', [900].TIME.YEAR := 2016, [900].TIME.MONTH := 9, [900].TIME.DAY := 26, [900].TIME.HOUR := 14, [900].TIME.MINUTE := 39, [900].TIME.SECOND := 50, [900].TIME.MICROSECOND := 992502, [900].EVENT := '2016/09/26   14:39:50   USER : PPS RESET FAULT BUTTON PRESSED', [901].TIME.YEAR := 2016, [901].TIME.MONTH := 9, [901].TIME.DAY := 26, [901].TIME.HOUR := 14, [901].TIME.MINUTE := 54, [901].TIME.MICROSECOND := 392490, [901].EVENT := '2016/09/26   14:54:00   USER : RESET FAULT BUTTON PRESSED', [902].TIME.YEAR := 2016, [902].TIME.MONTH := 9, [902].TIME.DAY := 26, [902].TIME.HOUR := 14, [902].TIME.MINUTE := 54, [902].TIME.SECOND := 8, [902].TIME.MICROSECOND := 892446, [902].EVENT := '2016/09/26   14:54:08   FAULT : WDT : Trigger Rate LOW', [903].TIME.YEAR := 2016, [903].TIME.MONTH := 9, [903].TIME.DAY := 26, [903].TIME.HOUR := 14, [903].TIME.MINUTE := 54, [903].TIME.SECOND := 16, [903].TIME.MICROSECOND := 992460, [903].EVENT := '2016/09/26   14:54:16   FAULT : TWB : Trigger Rate HIGH', [904].TIME.YEAR := 2016, [904].TIME.MONTH := 9, [904].TIME.DAY := 26, [904].TIME.HOUR := 14, [904].TIME.MINUTE := 54, [904].TIME.SECOND := 21, [904].TIME.MICROSECOND := 893000, [904].EVENT := '2016/09/26   14:54:21   USER : RESET FAULT BUTTON PRESSED', [905].TIME.YEAR := 2016, [905].TIME.MONTH := 9, [905].TIME.DAY := 26, [905].TIME.HOUR := 14, [905].TIME.MINUTE := 54, [905].TIME.SECOND := 25, [905].TIME.MICROSECOND := 692453, [905].EVENT := '2016/09/26   14:54:25   FAULT : TWB : Trigger Rate HIGH', [906].TIME.YEAR := 2016, [906].TIME.MONTH := 9, [906].TIME.DAY := 26, [906].TIME.HOUR := 14, [906].TIME.MINUTE := 54,
        [906].TIME.SECOND := 25, [906].TIME.MICROSECOND := 992446, [906].EVENT := '2016/09/26   14:54:25   FAULT : WDT : Trigger Rate LOW', [907].TIME.YEAR := 2016, [907].TIME.MONTH := 9, [907].TIME.DAY := 26, [907].TIME.HOUR := 14, [907].TIME.MINUTE := 54, [907].TIME.SECOND := 38, [907].TIME.MICROSECOND := 592489, [907].EVENT := '2016/09/26   14:54:38   USER : RESET FAULT BUTTON PRESSED', [908].TIME.YEAR := 2016, [908].TIME.MONTH := 9, [908].TIME.DAY := 26, [908].TIME.HOUR := 15, [908].TIME.MINUTE := 2, [908].TIME.SECOND := 21, [908].TIME.MICROSECOND := 892457, [908].EVENT := '2016/09/26   15:02:21   USER : CERTIFICATION MODE ENABLED', [909].TIME.YEAR := 2016, [909].TIME.MONTH := 9, [909].TIME.DAY := 26, [909].TIME.HOUR := 15, [909].TIME.MINUTE := 3, [909].TIME.SECOND := 20, [909].TIME.MICROSECOND := 192443, [909].EVENT := '2016/09/26   15:03:20   FAULT : WDT : Trigger Rate LOW', [910].TIME.YEAR := 2016, [910].TIME.MONTH := 9, [910].TIME.DAY := 26, [910].TIME.HOUR := 15, [910].TIME.MINUTE := 3, [910].TIME.SECOND := 25, [910].TIME.MICROSECOND := 692450, [910].EVENT := '2016/09/26   15:03:25   FAULT : TWB : Trigger Rate HIGH', [911].TIME.YEAR := 2016, [911].TIME.MONTH := 9, [911].TIME.DAY := 26, [911].TIME.HOUR := 15, [911].TIME.MINUTE := 3, [911].TIME.SECOND := 35, [911].TIME.MICROSECOND := 992487, [911].EVENT := '2016/09/26   15:03:35   USER : RESET FAULT BUTTON PRESSED', [912].TIME.YEAR := 2016, [912].TIME.MONTH := 9, [912].TIME.DAY := 26, [912].TIME.HOUR := 15, [912].TIME.MINUTE := 3, [912].TIME.SECOND := 59, [912].TIME.MICROSECOND := 892470, [912].EVENT := '2016/09/26   15:03:59   FAULT : TWB : Trigger Rate HIGH', [913].TIME.YEAR := 2016, [913].TIME.MONTH := 9, [913].TIME.DAY := 26, [913].TIME.HOUR := 15, [913].TIME.MINUTE := 4, [913].TIME.MICROSECOND := 192530, [913].EVENT := '2016/09/26   15:04:00   FAULT : WDT : Trigger Rate LOW', [914].TIME.YEAR := 2016, [914].TIME.MONTH := 9,
        [914].TIME.DAY := 26, [914].TIME.HOUR := 15, [914].TIME.MINUTE := 4, [914].TIME.SECOND := 20, [914].TIME.MICROSECOND := 692484, [914].EVENT := '2016/09/26   15:04:20   USER : RESET FAULT BUTTON PRESSED', [915].TIME.YEAR := 2016, [915].TIME.MONTH := 9, [915].TIME.DAY := 26, [915].TIME.HOUR := 15, [915].TIME.MINUTE := 4, [915].TIME.SECOND := 41, [915].TIME.MICROSECOND := 392893, [915].EVENT := '2016/09/26   15:04:41   FAULT : Self Test 2 Charge (B-A) LOW', [916].TIME.YEAR := 2016, [916].TIME.MONTH := 9, [916].TIME.DAY := 26, [916].TIME.HOUR := 15, [916].TIME.MINUTE := 4, [916].TIME.SECOND := 42, [916].TIME.MICROSECOND := 892829, [916].EVENT := '2016/09/26   15:04:42   FAULT : Self Test 2 Charge (A-B) LOW', [917].TIME.YEAR := 2016, [917].TIME.MONTH := 9, [917].TIME.DAY := 26, [917].TIME.HOUR := 15, [917].TIME.MINUTE := 5, [917].TIME.SECOND := 24, [917].TIME.MICROSECOND := 692910, [917].EVENT := '2016/09/26   15:05:24   USER : RESET FAULT BUTTON PRESSED', [918].TIME.YEAR := 2016, [918].TIME.MONTH := 9, [918].TIME.DAY := 26, [918].TIME.HOUR := 15, [918].TIME.MINUTE := 5, [918].TIME.SECOND := 39, [918].TIME.MICROSECOND := 992819, [918].EVENT := '2016/09/26   15:05:39   FAULT : Self Test 2 Charge (A-B) HIGH', [919].TIME.YEAR := 2016, [919].TIME.MONTH := 9, [919].TIME.DAY := 26, [919].TIME.HOUR := 15, [919].TIME.MINUTE := 5, [919].TIME.SECOND := 40, [919].TIME.MICROSECOND := 492883, [919].EVENT := '2016/09/26   15:05:40   FAULT : Self Test 2 Charge (B-A) HIGH', [920].TIME.YEAR := 2016, [920].TIME.MONTH := 9, [920].TIME.DAY := 26, [920].TIME.HOUR := 15, [920].TIME.MINUTE := 5, [920].TIME.SECOND := 40, [920].TIME.MICROSECOND := 992769, [920].EVENT := '2016/09/26   15:05:40   FAULT : Self Test 1 Charge (A-B) HIGH', [921].TIME.YEAR := 2016, [921].TIME.MONTH := 9, [921].TIME.DAY := 26, [921].TIME.HOUR := 15, [921].TIME.MINUTE := 5, [921].TIME.SECOND := 41,
        [921].TIME.MICROSECOND := 492786, [921].EVENT := '2016/09/26   15:05:41   FAULT : Self Test 1 Charge (B-A) HIGH', [922].TIME.YEAR := 2016, [922].TIME.MONTH := 9, [922].TIME.DAY := 26, [922].TIME.HOUR := 15, [922].TIME.MINUTE := 5, [922].TIME.SECOND := 41, [922].TIME.MICROSECOND := 493349, [922].EVENT := '2016/09/26   15:05:41   FAULT : Self Test 1 Charge (B-A) HIGH', [923].TIME.YEAR := 2016, [923].TIME.MONTH := 9, [923].TIME.DAY := 26, [923].TIME.HOUR := 15, [923].TIME.MINUTE := 6, [923].TIME.SECOND := 21, [923].TIME.MICROSECOND := 192488, [923].EVENT := '2016/09/26   15:06:21   USER : RESET FAULT BUTTON PRESSED', [924].TIME.YEAR := 2016, [924].TIME.MONTH := 9, [924].TIME.DAY := 26, [924].TIME.HOUR := 15, [924].TIME.MINUTE := 6, [924].TIME.SECOND := 41, [924].TIME.MICROSECOND := 692895, [924].EVENT := '2016/09/26   15:06:41   FAULT : Self Test 2 Charge (B-A) LOW', [925].TIME.YEAR := 2016, [925].TIME.MONTH := 9, [925].TIME.DAY := 26, [925].TIME.HOUR := 15, [925].TIME.MINUTE := 6, [925].TIME.SECOND := 41, [925].TIME.MICROSECOND := 693407, [925].EVENT := '2016/09/26   15:06:41   FAULT : Self Test 2 NO QAT DETECTED', [926].TIME.YEAR := 2016, [926].TIME.MONTH := 9, [926].TIME.DAY := 26, [926].TIME.HOUR := 15, [926].TIME.MINUTE := 6, [926].TIME.SECOND := 42, [926].TIME.MICROSECOND := 192781, [926].EVENT := '2016/09/26   15:06:42   FAULT : Self Test 1 Charge (A-B) LOW', [927].TIME.YEAR := 2016, [927].TIME.MONTH := 9, [927].TIME.DAY := 26, [927].TIME.HOUR := 15, [927].TIME.MINUTE := 6, [927].TIME.SECOND := 42, [927].TIME.MICROSECOND := 193368, [927].EVENT := '2016/09/26   15:06:42   FAULT : Self Test 1 NO QAT DETECTED', [928].TIME.YEAR := 2016, [928].TIME.MONTH := 9, [928].TIME.DAY := 26, [928].TIME.HOUR := 15, [928].TIME.MINUTE := 6, [928].TIME.SECOND := 42, [928].TIME.MICROSECOND := 692798, [928].EVENT := '2016/09/26   15:06:42   FAULT : Self Test 1 Charge (B-A) LOW', [929].TIME.YEAR := 2016, [929].TIME.MONTH := 9,
        [929].TIME.DAY := 26, [929].TIME.HOUR := 15, [929].TIME.MINUTE := 6, [929].TIME.SECOND := 43, [929].TIME.MICROSECOND := 192873, [929].EVENT := '2016/09/26   15:06:43   FAULT : Self Test 2 Charge (A-B) LOW', [930].TIME.YEAR := 2016, [930].TIME.MONTH := 9, [930].TIME.DAY := 26, [930].TIME.HOUR := 15, [930].TIME.MINUTE := 7, [930].TIME.MICROSECOND := 992919, [930].EVENT := '2016/09/26   15:07:00   USER : RESET FAULT BUTTON PRESSED', [931].TIME.YEAR := 2016, [931].TIME.MONTH := 9, [931].TIME.DAY := 26, [931].TIME.HOUR := 15, [931].TIME.MINUTE := 7, [931].TIME.SECOND := 11, [931].TIME.MICROSECOND := 392453, [931].EVENT := '2016/09/26   15:07:11   FAULT : QOW1 : Charge Outside Window Detected', [932].TIME.YEAR := 2016, [932].TIME.MONTH := 9, [932].TIME.DAY := 26, [932].TIME.HOUR := 15, [932].TIME.MINUTE := 7, [932].TIME.SECOND := 35, [932].TIME.MICROSECOND := 92487, [932].EVENT := '2016/09/26   15:07:35   USER : RESET FAULT BUTTON PRESSED', [933].TIME.YEAR := 2016, [933].TIME.MONTH := 9, [933].TIME.DAY := 26, [933].TIME.HOUR := 15, [933].TIME.MINUTE := 7, [933].TIME.SECOND := 41, [933].TIME.MICROSECOND := 992425, [933].EVENT := '2016/09/26   15:07:41   FAULT : Beam Charge HIGH', [934].TIME.YEAR := 2016, [934].TIME.MONTH := 9, [934].TIME.DAY := 26, [934].TIME.HOUR := 15, [934].TIME.MINUTE := 8, [934].TIME.SECOND := 1, [934].TIME.MICROSECOND := 892487, [934].EVENT := '2016/09/26   15:08:01   USER : RESET FAULT BUTTON PRESSED', [935].TIME.YEAR := 2016, [935].TIME.MONTH := 9, [935].TIME.DAY := 26, [935].TIME.HOUR := 15, [935].TIME.MINUTE := 8, [935].TIME.SECOND := 7, [935].TIME.MICROSECOND := 692453, [935].EVENT := '2016/09/26   15:08:07   FAULT : QOW1 : Charge Outside Window Detected', [936].TIME.YEAR := 2016, [936].TIME.MONTH := 9, [936].TIME.DAY := 26, [936].TIME.HOUR := 15, [936].TIME.MINUTE := 8, [936].TIME.SECOND := 7, [936].TIME.MICROSECOND := 792771,
        [936].EVENT := '2016/09/26   15:08:07   FAULT : Self Test 1 Charge (A-B) HIGH', [937].TIME.YEAR := 2016, [937].TIME.MONTH := 9, [937].TIME.DAY := 26, [937].TIME.HOUR := 15, [937].TIME.MINUTE := 8, [937].TIME.SECOND := 7, [937].TIME.MICROSECOND := 793344, [937].EVENT := '2016/09/26   15:08:07   FAULT : Self Test 1 B Baseline OUT OF RANGE', [938].TIME.YEAR := 2016, [938].TIME.MONTH := 9, [938].TIME.DAY := 26, [938].TIME.HOUR := 15, [938].TIME.MINUTE := 8, [938].TIME.SECOND := 7, [938].TIME.MICROSECOND := 992424, [938].EVENT := '2016/09/26   15:08:07   FAULT : Beam Charge LOW:', [939].TIME.YEAR := 2016, [939].TIME.MONTH := 9, [939].TIME.DAY := 26, [939].TIME.HOUR := 15, [939].TIME.MINUTE := 8, [939].TIME.SECOND := 7, [939].TIME.MICROSECOND := 992989, [939].EVENT := '2016/09/26   15:08:07   FAULT : Beam Baseline OUT OF RANGE', [940].TIME.YEAR := 2016, [940].TIME.MONTH := 9, [940].TIME.DAY := 26, [940].TIME.HOUR := 15, [940].TIME.MINUTE := 8, [940].TIME.SECOND := 8, [940].TIME.MICROSECOND := 292786, [940].EVENT := '2016/09/26   15:08:08   FAULT : Self Test 1 Charge (B-A) HIGH', [941].TIME.YEAR := 2016, [941].TIME.MONTH := 9, [941].TIME.DAY := 26, [941].TIME.HOUR := 15, [941].TIME.MINUTE := 8, [941].TIME.SECOND := 8, [941].TIME.MICROSECOND := 293356, [941].EVENT := '2016/09/26   15:08:08   FAULT : Self Test 1 Charge (B-A) HIGH', [942].TIME.YEAR := 2016, [942].TIME.MONTH := 9, [942].TIME.DAY := 26, [942].TIME.HOUR := 15, [942].TIME.MINUTE := 8, [942].TIME.SECOND := 8, [942].TIME.MICROSECOND := 293887, [942].EVENT := '2016/09/26   15:08:08   FAULT : Self Test 1 A Baseline OUT OF RANGE', [943].TIME.YEAR := 2016, [943].TIME.MONTH := 9, [943].TIME.DAY := 26, [943].TIME.HOUR := 15, [943].TIME.MINUTE := 8, [943].TIME.SECOND := 8, [943].TIME.MICROSECOND := 792817, [943].EVENT := '2016/09/26   15:08:08   FAULT : Self Test 2 Charge (A-B) HIGH', [944].TIME.YEAR := 2016, [944].TIME.MONTH := 9, [944].TIME.DAY := 26,
        [944].TIME.HOUR := 15, [944].TIME.MINUTE := 8, [944].TIME.SECOND := 8, [944].TIME.MICROSECOND := 793386, [944].EVENT := '2016/09/26   15:08:08   FAULT : Self Test 2 B Baseline OUT OF RANGE', [945].TIME.YEAR := 2016, [945].TIME.MONTH := 9, [945].TIME.DAY := 26, [945].TIME.HOUR := 15, [945].TIME.MINUTE := 8, [945].TIME.SECOND := 9, [945].TIME.MICROSECOND := 292886, [945].EVENT := '2016/09/26   15:08:09   FAULT : Self Test 2 Charge (B-A) HIGH', [946].TIME.YEAR := 2016, [946].TIME.MONTH := 9, [946].TIME.DAY := 26, [946].TIME.HOUR := 15, [946].TIME.MINUTE := 8, [946].TIME.SECOND := 9, [946].TIME.MICROSECOND := 293473, [946].EVENT := '2016/09/26   15:08:09   FAULT : Self Test 2 A Baseline OUT OF RANGE', [947].TIME.YEAR := 2016, [947].TIME.MONTH := 9, [947].TIME.DAY := 26, [947].TIME.HOUR := 15, [947].TIME.MINUTE := 8, [947].TIME.SECOND := 34, [947].TIME.MICROSECOND := 492487, [947].EVENT := '2016/09/26   15:08:34   USER : RESET FAULT BUTTON PRESSED', [948].TIME.YEAR := 2016, [948].TIME.MONTH := 9, [948].TIME.DAY := 26, [948].TIME.HOUR := 15, [948].TIME.MINUTE := 8, [948].TIME.SECOND := 42, [948].TIME.MICROSECOND := 692374, [948].EVENT := '2016/09/26   15:08:42   FAULT : Self Test 2 Charge (B-A) LOW', [949].TIME.YEAR := 2016, [949].TIME.MONTH := 9, [949].TIME.DAY := 26, [949].TIME.HOUR := 15, [949].TIME.MINUTE := 8, [949].TIME.SECOND := 42, [949].TIME.MICROSECOND := 693006, [949].EVENT := '2016/09/26   15:08:42   FAULT : TWB : Trigger Rate HIGH', [950].TIME.YEAR := 2016, [950].TIME.MONTH := 9, [950].TIME.DAY := 26, [950].TIME.HOUR := 15, [950].TIME.MINUTE := 8, [950].TIME.SECOND := 42, [950].TIME.MICROSECOND := 693502, [950].EVENT := '2016/09/26   15:08:42   FAULT : QOW1 : Charge Outside Window Detected', [951].TIME.YEAR := 2016, [951].TIME.MONTH := 9, [951].TIME.DAY := 26, [951].TIME.HOUR := 15, [951].TIME.MINUTE := 8, [951].TIME.SECOND := 42, [951].TIME.MICROSECOND := 694050,
        [951].EVENT := '2016/09/26   15:08:42   USER : CERTIFICATION MODE DISABLED', [952].TIME.YEAR := 2016, [952].TIME.MONTH := 9, [952].TIME.DAY := 26, [952].TIME.HOUR := 15, [952].TIME.MINUTE := 8, [952].TIME.SECOND := 43, [952].TIME.MICROSECOND := 192447, [952].EVENT := '2016/09/26   15:08:43   FAULT : WDT : Trigger Rate LOW', [953].TIME.YEAR := 2016, [953].TIME.MONTH := 9, [953].TIME.DAY := 26, [953].TIME.HOUR := 15, [953].TIME.MINUTE := 9, [953].TIME.SECOND := 2, [953].TIME.MICROSECOND := 392463, [953].EVENT := '2016/09/26   15:09:02   USER : CERTIFICATION MODE ENABLED', [954].TIME.YEAR := 2016, [954].TIME.MONTH := 9, [954].TIME.DAY := 26, [954].TIME.HOUR := 15, [954].TIME.MINUTE := 9, [954].TIME.SECOND := 6, [954].TIME.MICROSECOND := 392492, [954].EVENT := '2016/09/26   15:09:06   USER : RESET FAULT BUTTON PRESSED', [955].TIME.YEAR := 2016, [955].TIME.MONTH := 9, [955].TIME.DAY := 26, [955].TIME.HOUR := 15, [955].TIME.MINUTE := 11, [955].TIME.SECOND := 4, [955].TIME.MICROSECOND := 792494, [955].EVENT := '2016/09/26   15:11:04   USER : RESET ALL KEY SWITCH ENABLED', [956].TIME.YEAR := 2016, [956].TIME.MONTH := 9, [956].TIME.DAY := 26, [956].TIME.HOUR := 15, [956].TIME.MINUTE := 11, [956].TIME.SECOND := 5, [956].TIME.MICROSECOND := 592924, [956].EVENT := '2016/09/26   15:11:05   USER : RESET ALL BUTTON PRESSED', [957].TIME.YEAR := 2016, [957].TIME.MONTH := 9, [957].TIME.DAY := 26, [957].TIME.HOUR := 15, [957].TIME.MINUTE := 13, [957].TIME.SECOND := 11, [957].TIME.MICROSECOND := 392937, [957].EVENT := '2016/09/26   15:13:11   USER : PPS RESET FAULT BUTTON PRESSED', [958].TIME.YEAR := 2016, [958].TIME.MONTH := 9, [958].TIME.DAY := 26, [958].TIME.HOUR := 15, [958].TIME.MINUTE := 58, [958].TIME.SECOND := 21, [958].TIME.MICROSECOND := 92474, [958].EVENT := '2016/09/26   15:58:21   FAULT : Booster Ring Accumulation HIGH', [959].TIME.YEAR := 2016, [959].TIME.MONTH := 9, [959].TIME.DAY := 26,
        [959].TIME.HOUR := 16, [959].TIME.MINUTE := 7, [959].TIME.SECOND := 33, [959].TIME.MICROSECOND := 392450, [959].EVENT := '2016/09/26   16:07:33   FAULT : Booster Ring Accumulation HIGH', [960].TIME.YEAR := 2016, [960].TIME.MONTH := 9, [960].TIME.DAY := 26, [960].TIME.HOUR := 16, [960].TIME.MINUTE := 7, [960].TIME.SECOND := 33, [960].TIME.MICROSECOND := 393054, [960].EVENT := '2016/09/26   16:07:33   USER : RESET FAULT BUTTON PRESSED', [961].TIME.YEAR := 2016, [961].TIME.MONTH := 9, [961].TIME.DAY := 26, [961].TIME.HOUR := 16, [961].TIME.MINUTE := 12, [961].TIME.SECOND := 2, [961].TIME.MICROSECOND := 792492, [961].EVENT := '2016/09/26   16:12:02   USER : RESET FAULT BUTTON PRESSED', [962].TIME.YEAR := 2016, [962].TIME.MONTH := 9, [962].TIME.DAY := 26, [962].TIME.HOUR := 16, [962].TIME.MINUTE := 12, [962].TIME.SECOND := 2, [962].TIME.MICROSECOND := 892441, [962].EVENT := '2016/09/26   16:12:02   FAULT : Booster Ring Accumulation HIGH', [963].TIME.YEAR := 2016, [963].TIME.MONTH := 9, [963].TIME.DAY := 26, [963].TIME.HOUR := 16, [963].TIME.MINUTE := 12, [963].TIME.SECOND := 14, [963].TIME.MICROSECOND := 592493, [963].EVENT := '2016/09/26   16:12:14   USER : RESET FAULT BUTTON PRESSED', [964].TIME.YEAR := 2016, [964].TIME.MONTH := 9, [964].TIME.DAY := 26, [964].TIME.HOUR := 16, [964].TIME.MINUTE := 12, [964].TIME.SECOND := 17, [964].TIME.MICROSECOND := 692492, [964].EVENT := '2016/09/26   16:12:17   USER : RESET FAULT BUTTON PRESSED', [965].TIME.YEAR := 2016, [965].TIME.MONTH := 9, [965].TIME.DAY := 26, [965].TIME.HOUR := 16, [965].TIME.MINUTE := 12, [965].TIME.SECOND := 34, [965].TIME.MICROSECOND := 492642, [965].EVENT := '2016/09/26   16:12:34   USER : RESET ALL KEY SWITCH ENABLED', [966].TIME.YEAR := 2016, [966].TIME.MONTH := 9, [966].TIME.DAY := 26, [966].TIME.HOUR := 16, [966].TIME.MINUTE := 12, [966].TIME.SECOND := 36, [966].TIME.MICROSECOND := 492498,
        [966].EVENT := '2016/09/26   16:12:36   USER : RESET ALL BUTTON PRESSED', [967].TIME.YEAR := 2016, [967].TIME.MONTH := 9, [967].TIME.DAY := 26, [967].TIME.HOUR := 16, [967].TIME.MINUTE := 12, [967].TIME.SECOND := 54, [967].TIME.MICROSECOND := 992496, [967].EVENT := '2016/09/26   16:12:54   USER : RESET ALL KEY SWITCH ENABLED', [968].TIME.YEAR := 2016, [968].TIME.MONTH := 9, [968].TIME.DAY := 26, [968].TIME.HOUR := 16, [968].TIME.MINUTE := 12, [968].TIME.SECOND := 55, [968].TIME.MICROSECOND := 593016, [968].EVENT := '2016/09/26   16:12:55   USER : RESET ALL BUTTON PRESSED', [969].TIME.YEAR := 2016, [969].TIME.MONTH := 9, [969].TIME.DAY := 26, [969].TIME.HOUR := 17, [969].TIME.MINUTE := 24, [969].TIME.SECOND := 26, [969].TIME.MICROSECOND := 692442, [969].EVENT := '2016/09/26   17:24:26   FAULT : WDT : Trigger Rate LOW', [970].TIME.YEAR := 2016, [970].TIME.MONTH := 9, [970].TIME.DAY := 27, [970].TIME.HOUR := 8, [970].TIME.MINUTE := 6, [970].TIME.SECOND := 52, [970].TIME.MICROSECOND := 492498, [970].EVENT := '2016/09/27   08:06:52   USER : PPS RESET FAULT BUTTON PRESSED', [971].TIME.YEAR := 2016, [971].TIME.MONTH := 9, [971].TIME.DAY := 27, [971].TIME.HOUR := 8, [971].TIME.MINUTE := 7, [971].TIME.SECOND := 25, [971].TIME.MICROSECOND := 292498, [971].EVENT := '2016/09/27   08:07:25   USER : PPS RESET FAULT BUTTON PRESSED', [972].TIME.YEAR := 2016, [972].TIME.MONTH := 9, [972].TIME.DAY := 27, [972].TIME.HOUR := 8, [972].TIME.MINUTE := 7, [972].TIME.SECOND := 26, [972].TIME.MICROSECOND := 192522, [972].EVENT := '2016/09/27   08:07:26   USER : PPS RESET FAULT BUTTON PRESSED', [973].TIME.YEAR := 2016, [973].TIME.MONTH := 9, [973].TIME.DAY := 27, [973].TIME.HOUR := 8, [973].TIME.MINUTE := 7, [973].TIME.SECOND := 26, [973].TIME.MICROSECOND := 592501, [973].EVENT := '2016/09/27   08:07:26   USER : PPS RESET FAULT BUTTON PRESSED', [974].TIME.YEAR := 2016, [974].TIME.MONTH := 9, [974].TIME.DAY := 27,
        [974].TIME.HOUR := 8, [974].TIME.MINUTE := 7, [974].TIME.SECOND := 26, [974].TIME.MICROSECOND := 992505, [974].EVENT := '2016/09/27   08:07:26   USER : PPS RESET FAULT BUTTON PRESSED', [975].TIME.YEAR := 2016, [975].TIME.MONTH := 9, [975].TIME.DAY := 27, [975].TIME.HOUR := 8, [975].TIME.MINUTE := 7, [975].TIME.SECOND := 27, [975].TIME.MICROSECOND := 292502, [975].EVENT := '2016/09/27   08:07:27   USER : PPS RESET FAULT BUTTON PRESSED', [976].TIME.YEAR := 2016, [976].TIME.MONTH := 9, [976].TIME.DAY := 27, [976].TIME.HOUR := 8, [976].TIME.MINUTE := 24, [976].TIME.SECOND := 8, [976].TIME.MICROSECOND := 292504, [976].EVENT := '2016/09/27   08:24:08   USER : PPS RESET FAULT BUTTON PRESSED', [977].TIME.YEAR := 2016, [977].TIME.MONTH := 9, [977].TIME.DAY := 27, [977].TIME.HOUR := 9, [977].TIME.MINUTE := 5, [977].TIME.SECOND := 9, [977].TIME.MICROSECOND := 892488, [977].EVENT := '2016/09/27   09:05:09   USER : RESET FAULT BUTTON PRESSED', [978].TIME.YEAR := 2016, [978].TIME.MONTH := 9, [978].TIME.DAY := 27, [978].TIME.HOUR := 9, [978].TIME.MINUTE := 5, [978].TIME.SECOND := 27, [978].TIME.MICROSECOND := 92497, [978].EVENT := '2016/09/27   09:05:27   USER : RESET ALL KEY SWITCH ENABLED', [979].TIME.YEAR := 2016, [979].TIME.MONTH := 9, [979].TIME.DAY := 27, [979].TIME.HOUR := 9, [979].TIME.MINUTE := 5, [979].TIME.SECOND := 28, [979].TIME.MICROSECOND := 292495, [979].EVENT := '2016/09/27   09:05:28   USER : RESET ALL BUTTON PRESSED', [980].TIME.YEAR := 2016, [980].TIME.MONTH := 9, [980].TIME.DAY := 27, [980].TIME.HOUR := 9, [980].TIME.MINUTE := 8, [980].TIME.SECOND := 57, [980].TIME.MICROSECOND := 892891, [980].EVENT := '2016/09/27   09:08:57   FAULT : Self Test 2 Charge (B-A) HIGH', [981].TIME.YEAR := 2016, [981].TIME.MONTH := 9, [981].TIME.DAY := 27, [981].TIME.HOUR := 9, [981].TIME.MINUTE := 8, [981].TIME.SECOND := 57, [981].TIME.MICROSECOND := 893409,
        [981].EVENT := '2016/09/27   09:08:57   FAULT : Self Test 2 A Baseline OUT OF RANGE', [982].TIME.YEAR := 2016, [982].TIME.MONTH := 9, [982].TIME.DAY := 27, [982].TIME.HOUR := 9, [982].TIME.MINUTE := 8, [982].TIME.SECOND := 57, [982].TIME.MICROSECOND := 894030, [982].EVENT := '2016/09/27   09:08:57   FAULT : QOW1 : Charge Outside Window Detected', [983].TIME.YEAR := 2016, [983].TIME.MONTH := 9, [983].TIME.DAY := 27, [983].TIME.HOUR := 9, [983].TIME.MINUTE := 8, [983].TIME.SECOND := 58, [983].TIME.MICROSECOND := 92432, [983].EVENT := '2016/09/27   09:08:58   FAULT : Beam Charge LOW:', [984].TIME.YEAR := 2016, [984].TIME.MONTH := 9, [984].TIME.DAY := 27, [984].TIME.HOUR := 9, [984].TIME.MINUTE := 8, [984].TIME.SECOND := 58, [984].TIME.MICROSECOND := 92997, [984].EVENT := '2016/09/27   09:08:58   FAULT : Beam Baseline OUT OF RANGE', [985].TIME.YEAR := 2016, [985].TIME.MONTH := 9, [985].TIME.DAY := 27, [985].TIME.HOUR := 9, [985].TIME.MINUTE := 8, [985].TIME.SECOND := 58, [985].TIME.MICROSECOND := 392773, [985].EVENT := '2016/09/27   09:08:58   FAULT : Self Test 1 Charge (A-B) HIGH', [986].TIME.YEAR := 2016, [986].TIME.MONTH := 9, [986].TIME.DAY := 27, [986].TIME.HOUR := 9, [986].TIME.MINUTE := 8, [986].TIME.SECOND := 58, [986].TIME.MICROSECOND := 393412, [986].EVENT := '2016/09/27   09:08:58   FAULT : Self Test 1 B Baseline OUT OF RANGE', [987].TIME.YEAR := 2016, [987].TIME.MONTH := 9, [987].TIME.DAY := 27, [987].TIME.HOUR := 9, [987].TIME.MINUTE := 8, [987].TIME.SECOND := 58, [987].TIME.MICROSECOND := 892787, [987].EVENT := '2016/09/27   09:08:58   FAULT : Self Test 1 Charge (B-A) HIGH', [988].TIME.YEAR := 2016, [988].TIME.MONTH := 9, [988].TIME.DAY := 27, [988].TIME.HOUR := 9, [988].TIME.MINUTE := 8, [988].TIME.SECOND := 58, [988].TIME.MICROSECOND := 893353, [988].EVENT := '2016/09/27   09:08:58   FAULT : Self Test 1 Charge (B-A) HIGH', [989].TIME.YEAR := 2016, [989].TIME.MONTH := 9, [989].TIME.DAY := 27,
        [989].TIME.HOUR := 9, [989].TIME.MINUTE := 8, [989].TIME.SECOND := 58, [989].TIME.MICROSECOND := 893882, [989].EVENT := '2016/09/27   09:08:58   FAULT : Self Test 1 A Baseline OUT OF RANGE', [990].TIME.YEAR := 2016, [990].TIME.MONTH := 9, [990].TIME.DAY := 27, [990].TIME.HOUR := 9, [990].TIME.MINUTE := 8, [990].TIME.SECOND := 59, [990].TIME.MICROSECOND := 392873, [990].EVENT := '2016/09/27   09:08:59   FAULT : Self Test 2 Charge (A-B) HIGH', [991].TIME.YEAR := 2016, [991].TIME.MONTH := 9, [991].TIME.DAY := 27, [991].TIME.HOUR := 9, [991].TIME.MINUTE := 8, [991].TIME.SECOND := 59, [991].TIME.MICROSECOND := 393392, [991].EVENT := '2016/09/27   09:08:59   FAULT : Self Test 2 B Baseline OUT OF RANGE', [992].TIME.YEAR := 2016, [992].TIME.MONTH := 9, [992].TIME.DAY := 27, [992].TIME.HOUR := 9, [992].TIME.MINUTE := 9, [992].TIME.SECOND := 3, [992].TIME.MICROSECOND := 692489, [992].EVENT := '2016/09/27   09:09:03   USER : RESET FAULT BUTTON PRESSED', [993].TIME.YEAR := 2016, [993].TIME.MONTH := 9, [993].TIME.DAY := 27, [993].TIME.HOUR := 9, [993].TIME.MINUTE := 45, [993].TIME.SECOND := 19, [993].TIME.MICROSECOND := 92429, [993].EVENT := '2016/09/27   09:45:19   FAULT : Beam Charge HIGH', [994].TIME.YEAR := 2016, [994].TIME.MONTH := 9, [994].TIME.DAY := 27, [994].TIME.HOUR := 9, [994].TIME.MINUTE := 45, [994].TIME.SECOND := 19, [994].TIME.MICROSECOND := 592437, [994].EVENT := '2016/09/27   09:45:19   FAULT : Storage Ring Accumulation HIGH', [995].TIME.YEAR := 2016, [995].TIME.MONTH := 9, [995].TIME.DAY := 27, [995].TIME.HOUR := 9, [995].TIME.MINUTE := 45, [995].TIME.SECOND := 29, [995].TIME.MICROSECOND := 292718, [995].EVENT := '2016/09/27   09:45:29   FAULT : Storage Ring Accumulation HIGH', [996].TIME.YEAR := 2016, [996].TIME.MONTH := 9, [996].TIME.DAY := 27, [996].TIME.HOUR := 9, [996].TIME.MINUTE := 45, [996].TIME.SECOND := 30, [996].TIME.MICROSECOND := 992905,
        [996].EVENT := '2016/09/27   09:45:30   USER : RESET FAULT BUTTON PRESSED', [997].TIME.YEAR := 2016, [997].TIME.MONTH := 9, [997].TIME.DAY := 27, [997].TIME.HOUR := 9, [997].TIME.MINUTE := 45, [997].TIME.SECOND := 35, [997].TIME.MICROSECOND := 892720, [997].EVENT := '2016/09/27   09:45:35   FAULT : Storage Ring Accumulation HIGH', [998].TIME.YEAR := 2016, [998].TIME.MONTH := 9, [998].TIME.DAY := 27, [998].TIME.HOUR := 9, [998].TIME.MINUTE := 45, [998].TIME.SECOND := 38, [998].TIME.MICROSECOND := 692999, [998].EVENT := '2016/09/27   09:45:38   USER : RESET FAULT BUTTON PRESSED', [999].TIME.YEAR := 2016, [999].TIME.MONTH := 9, [999].TIME.DAY := 27, [999].TIME.HOUR := 9, [999].TIME.MINUTE := 46, [999].TIME.SECOND := 4, [999].TIME.MICROSECOND := 392498, [999].EVENT := '2016/09/27   09:46:04   USER : RESET FAULT BUTTON PRESSED'); {access Read Only}
   ELog_Size : DINT := 21858; {access Read Only}
   Enext : BOOL;
   Enextons : BOOL;
   Epage : EVENT[30];
   Eprev : BOOL;
   Eprevons : BOOL;
   Eupdate : BOOL;
   evnum : DINT := 1;
   fault_1 : BOOL := 1; {access Read Only}
   fault_10 : BOOL := 1; {access Read Only}
   fault_11 : BOOL := 1; {access Read Only}
   fault_12 : BOOL := 1; {access Read Only}
   fault_13 : BOOL := 1; {access Read Only}
   fault_14 : BOOL := 1; {access Read Only}
   fault_15 : BOOL := 1; {access Read Only}
   fault_16 : BOOL := 1; {access Read Only}
   fault_17 : BOOL := 1; {access Read Only}
   fault_18 : BOOL; {access Read Only}
   fault_19 : BOOL; {access Read Only}
   fault_2 : BOOL := 1; {access Read Only}
   fault_20 : BOOL; {access Read Only}
   fault_21 : BOOL; {access Read Only}
   fault_22 : BOOL := 1; {access Read Only}
   fault_23 : BOOL := 1; {access Read Only}
   fault_3 : BOOL := 1; {access Read Only}
   fault_4 : BOOL := 1; {access Read Only}
   fault_5 : BOOL := 1; {access Read Only}
   fault_6 : BOOL := 1; {access Read Only}
   fault_7 : BOOL := 1; {access Read Only}
   fault_8 : BOOL := 1; {access Read Only}
   fault_9 : BOOL := 1; {access Read Only}
   fault_string : STRING := 'FAULT : Beam Baseline OUT OF RANGE'; {access Read Only}
   message : STRING[35] := ([0] := 'FAULT : Self Test 2 Charge (A-B) HIGH', [1] := 'FAULT : Self Test 2 Charge (A-B) LOW', [2] := 'FAULT : Self Test 2 B Baseline OUT OF RANGE', [3] := 'FAULT : Self Test 2 Charge (B-A) HIGH', [4] := 'FAULT : Self Test 2 Charge (B-A) LOW', [5] := 'FAULT : Self Test 2 A Baseline OUT OF RANGE', [6] := 'FAULT : Self Test 1 Charge (A-B) HIGH', [7] := 'FAULT : Self Test 1 Charge (A-B) LOW', [8] := 'FAULT : Self Test 1 B Baseline OUT OF RANGE', [9] := 'FAULT : Self Test 1 Charge (B-A) HIGH', [10] := 'FAULT : Self Test 1 Charge (B-A) LOW', [11] := 'FAULT : Self Test 1 A Baseline OUT OF RANGE', [12] := 'FAULT : Self Test 1 NO QAT DETECTED', [13] := 'FAULT : Beam Charge LOW:', [14] := 'FAULT : Beam Charge HIGH', [15] := 'FAULT : Beam Baseline OUT OF RANGE', [16] := 'FAULT : Booster Ring Accumulation HIGH', [17] := 'FAULT : Storage Ring Accumulation HIGH', [18] := 'FAULT : WDT : Trigger Rate LOW', [19] := 'FAULT : TWB : Trigger Rate HIGH', [20] := 'FAULT : QOW1 : Charge Outside Window Detected', [21] := 'FAULT : Self Test 2 NO QAT DETECTED', [22] := 'USER : CERTIFICATION MODE ENABLED', [23] := 'USER : CERTIFICATION MODE DISABLED', [24] := 'USER : TIMING MODE ENABLED', [25] := 'USER : TIMING MODE DISABLED', [26] := 'USER : SAFETY SHUTTERS OPENED', [27] := 'USER : SAFETY SHUTTERS CLOSED', [28] := 'USER : RESET FAULT BUTTON PRESSED', [29] := 'USER : RESET ALL KEY SWITCH ENABLED', [30] := 'USER : RESET ALL BUTTON PRESSED', [31] := 'USER : PPS RESET FAULT BUTTON PRESSED', [32] := 'USER : BYPASS KEY SET TO ENABLE', [33] := 'USER : BYPASS KEY SET TO DISABLE'); {constant, access Read Only}
   nada : STRING := '0'; {constant, access Read Only}
   slash : STRING := '/'; {constant, access Read Only}
   space : STRING := '   '; {constant, access Read Only}
   str : STRING := '04'; {access Read Only}
END_VAR
